M2VGwvK0duS1QvaFp5aC80ZWJvLytIbktYL2k2Q28vNHFlcVArT3BLNy9ncGFiLzRLVGwvK0lsSjMvaG8rVi80NmRyUCtkc2J6L25hNjkvNTJ2dnYrYnJMdi9uckc2LzVhc3VQK1ZyN3YvbWE2My81KzJ3LytjdE1EL203ZSsvNXF6dlArTm9hYi9qS09uLzVtenQvK2JzYlQvazZ1dS80K21xLytRcWF2L2tLbXQvNUdyclArZ3Riei9sYWlxLzVLcHFQK0xvS1gvajZTbC81R2hvUCtQbzZQL2xhcXIvNU9wcWYrVHA2ai9rcXF0LzVPa3BmK0ttSmYvbkdOdi83SkdWdjl2ZjRYL2phS2YvNG1aa3YrUG82UC9pcCtmLzRxZW9mK1BwcUgvaFptVy80U1psZitIbDVUL2dwS1EvNGVVa3Y5Z2NYYi9sSk4rL3lVZkYvOEtEUW4vSkN3bS8wOWRVdjlYWlZyL1dHZGMvMTlzWHY5ZGFGMy9YV2RnLzF4cFlmOWRiR1AvWTNKci8yVjBhLzlvYzJ2L2FYVnUvMlp6YnY5cGMyLy9ibmgwLzJ4M2N2OXJlSEwvYjMxNi8zcUZndjkyZ24vL2M0Ri8vM0Y5ZlA5eWYzLy9jbjE3LzNSK2VmOTZnNEgvZTRXRy8zaUhndjk3aUlUL2Y0MkcvMytLaFArRWtJMy9pSk9NLzRlVGp2K09tcEgvZ1k2SC80T1NqLzk2allYL2ZaS0svNE9YanYrR2xvdi9mbzJILzM2T2hmOTlrSVQvZll1Qy8zeU1nUDk0aVlIL2VZbUQvMzJLaC85K2pZTC9kNHFBLzNxS2hmOTNoWVAvZVllQi8zV0dnUDkyaUlIL2NvZCsvM2FKZ1A5Mmk0SC9lWWVDLzN1S2hmOTNpNFAvams5Vi84TkVVLytFaW9UL2ZJNkUvM3lQaXY5N2tJci9lNUdPLzRLVmpQOS9rNDcvZ0pLUi8zK1dqZitEbFkzL2dKYU4vMzZWanYrYnBKbi9JU1FlL3hnZkdmOVJZVlQvWlhSby8yVjBhLzluZDIvL2JIbHUvMnQ3Y3Y5dWZIVC9iWHh5LzIxK2RmOXdoSG4vYzRWOS8zZUdnZjk0aVlUL2VJbUYvM2VHZy8rQWpZMy9ncEtOLzRPV2tmK0dtWlgvaUp5Vi80YVlsZitKbTZEL2taK2MvNUdmblArUW5aMy9rcVdoLzVLam52K1ZwS1gvbTZ5cy81cXJxditoc0svL25xK3QvNlN6c3YrcXZyei9vYlN4LzZLNHNmK2d1YlAvcHIyMS81MjNzUCtpdTdiL3BicTAvNWV0cGYrV3JLVC9rYVdhLzVDaWxQK01uSkgvaFpxSS80S1JnditBa1lYL2ZJNkQvM3VPZ3Y5M2kzMy9kb2QrLzNPRWV2OXdnWFQvY1gxMy8yMThkUDl0Zm5UL2JYdHkvMnA1YnY5cGQyMy9ablZyLzJSemFmOW5kR3ovbTBwUi83UXpRdjlqYTJML1gyMWovMkJzWWY5Z2EyRC9YbXRoLzExclgvOWVhMTcvVzJ0Yy8xbG9YZjlYWmx6L1ZtWlovMXBYVy84bUp5VC9TbFpJLzFCZVUvOW9kR3IvYW5acS8yaDViLzlyZUcvL2JYcHkvMng4ZGY5c2dYai9jNFY2LzI1L2QvOXhnbnovZDRTQS8zdUhnUDk2aW9iL2U1Q0ovNE9ZbGYrRWxZNy9ncFdOLzRlWWxQK0psNUwvajZLZC80dVptditTcGFiL242MnMvNXlycWYrWnJhdi9tcW1uLzVlb3B2K2FyYXYvbks2eC82NjV1ditpczZ6L3FMdTIvNmk5dGYrcndyci9xTDYxLzZTNXN2K2t1YmovcHJ5NC82ZThzZitndHFyL21LdWgvNU9tb1ArT281di9qNkdXLzQraW1QK0dtSTcvaHBxTS80Q1BoUDk4aTRQL2VZcCsvM3FLZ3Y5NWg0TC9jWUY4LzNPRWVmOXdnbmYvYTNwei8yeDhkUDlyZDIzL2FYaHQvMmw3YnY5cGRtMy9hSFJyLzJaMmEvOWlkR2ovazB4Ui82NDRSdjlqYW1IL1luQmsvMkZ1WXY5ZWJXTC9YMjVpLzE1dFl2OWRiR0QvVzJwZi8xdHFYZjlhYWx2L1NFbzcvMHhLUC85ZGFWLy9UbHROLzJSd2FQOW9lVy8vYUhsdi8ydDNiLzl2ZjNQL2EzMXkvMjJBZHY5dGczci9kSVoyLzN1SGZmOTBoSHIvZG9pQi8zMlBpdjkzaW9iL2daV08vNEdZai8rRm1KRC9pcHlYLzRtY2xQK05vSnIvaTZXaS81Q2lvLytTcEtEL2w3Q3EvNXkwci8raXRySC9vcld1LzZXMHIvK2pyN0gvcExXdi82aTR0UCtydWJmL3FidTUvNnEvdVArdHdMYi9xNyswLzZXOHRQK3B3TFQvbjd5dS82SytzUCtsdUs3L2w2cWcvNHlobVArSm41SC9qNktVLzRTV2pmK0dtbzcvZ0pHRS80R09nLzk2aW43L2Q0Wi8vM2lLZ1A5eWhYMy9jSU4zLzNHQ2R2OXRmM0wvYW4xdi8ybDZidjlwZVczL2FYbHUvMmQwYXY5bWRXdi9hWGh0LzJaMWF2OWtjMmovakV0Ui83SXVRUDlxWm1EL1lXOWwvMTl3WlA5ZmJHUC9YbXhrLzExc1lmOWNhVi8vVzJsZS8xcHBYSGdcdTAwM2QiLCJfdGVhY2hNZXRob2QiOnsiX21ldGhvZFR5cGUiOiJBVVRPTUFUSUMifSwiX2lzSWdub3JlU25hcHNob3RQb3NpdGlvbiI6ZmFsc2UsIl9pc0F1dG9tYXRpY01vdmUiOnRydWUsIl9pc0lnbm9yZVJvdGF0aW9uIjpmYWxzZX0=]); state(isChildrenLocked=true)
        URCap Boucle de la localisation de caméra (Robotiq_Wrist_Camera, Robotiq Inc.)
          MoveL speed 80 mm/s, acceleration 50 mm/s^2 (useActiveTCP=true) feature=Calib_1
            Waypoint approche: motionParameters(jointSpeed=1.047198 jointAcceleration=1.396263 cartesianSpeed=0.4 cartesianAcceleration=0.508); TCP in base x=-127.51 y=-324.345 z=215.094 mm, rx=-2.2625 ry=-2.1587 rz=0.0418 rad; joints [-89.286, -99.558, -104.123, -65.824, 88.206, -266.16] deg; feature pose in base x=-115.28 y=-376.355 z=-47.016 mm, rx=2.2478 ry=2.1911 rz=0 rad
            Waypoint recup: motionParameters(jointSpeed=1.047198 jointAcceleration=1.396263 cartesianSpeed=0.15 cartesianAcceleration=0.08); TCP in base x=-120.621 y=-324.408 z=153.783 mm, rx=-2.2059 ry=-2.2161 rz=0.0393 rad; joints [-88.063, -107.147, -113.625, -48.801, 88.216, -267.906] deg
            URCap Main (Robotiq_Grippers, Robotiq Inc.) dataModel(position=55.0, force=0.0, speed=0.0, positionInDouble=55.0, forceInDouble=0.0, speedInDouble=0.0, slaveIds=[9], blocking=true)
            Waypoint approche: motionParameters(jointSpeed=1.047198 jointAcceleration=1.396263 cartesianSpeed=0.15 cartesianAcceleration=0.08); TCP in base x=-127.51 y=-324.345 z=215.094 mm, rx=-2.2625 ry=-2.1587 rz=0.0418 rad; joints [-89.286, -99.558, -104.123, -65.824, 88.206, -266.16] deg
            Waypoint post_prise: motionParameters(jointSpeed=1.047198 jointAcceleration=1.396263 cartesianSpeed=0.25 cartesianAcceleration=1.2); TCP in base x=-119.842 y=-320.203 z=232.501 mm, rx=3.123 ry=-0.1407 rz=0.0686 rad; joints [-89.094, -96.9, -102.497, -69.534, 92.351, -173.46] deg; feature pose in base x=-181.238 y=-310.931 z=-23.576 mm, rx=3.1384 ry=-0.0927 rz=0.0029 rad
            var_1 := False
          MoveJ speed 80 deg/s, acceleration 80 deg/s^2 (useActiveTCP=true) feature=Base
            Waypoint pro_placer: TCP in base x=-107.3 y=-316.96 z=388.086 mm, rx=2.2531 ry=2.1366 rz=-0.0153 rad; joints [-86.259, -95.495, -61.717, -110.755, 90.787, -262.768] deg
            Waypoint Placer_rebus: TCP in base x=-499.436 y=-158.136 z=389.522 mm, rx=-1.535 ry=-1.7186 rz=0.8921 rad; joints [-143.293, -133.833, -33.792, -50.34, 63.066, -342.955] deg
            URCap Main (Robotiq_Grippers, Robotiq Inc.) dataModel(position=0.0, force=0.0, speed=0.0, positionInDouble=0.0, forceInDouble=0.0, speedInDouble=0.0, slaveIds=[9], blocking=true)
            Waypoint PointPassage_6: TCP in base x=-341.675 y=-103.087 z=420.535 mm, rx=-1.8218 ry=-2.4283 rz=-0.0315 rad; joints [-140.176, -106.769, -36.81, -126.166, 83.655, -336.031] deg
            Waypoint retour_securise: TCP in base x=-134.176 y=-179.969 z=442.128 mm, rx=-2.2471 ry=-2.1697 rz=0.0496 rad; joints [-90.577, -75.287, -61.755, -132.356, 88.017, -268.12] deg
        URCap Si aucun objet n’est détecté par la caméra (Robotiq_Wrist_Camera, Robotiq Inc.)
          'Optionnel'
